FUNCTION_BLOCK NullItem IMPLEMENTS I_Base
VAR
END_VAR

END_FUNCTION_BLOCK

(* stored: Version 1.1.0.1, ProductVersion 3.1.4026.18
   POU NullItem: Id {69305bfe-9891-4a94-b77e-852628667a5b}, SpecialFunc None *)
